{attribute 'linkalways'} 
{attribute 'no_explicit_call' := 'This FB is a CLASS and must be accessed using methods or properties'}
{attribute 'enable_dynamic_creation'}
FUNCTION_BLOCK ReleaseAxisCommand EXTENDS NciCommand
VAR
	_fb : CfgReconfigAxis;
	_axisId : UDINT;
	_timeout : TIME;
END_VAR

METHOD FB_init : BOOL
VAR_INPUT
	bInitRetains : BOOL; // if TRUE, the retain variables are initialized (warm start / cold start)
	bInCopyCode : BOOL;  // if TRUE, the instance afterwards gets moved into the copy code (online change)
	axis : I_Axis;
	timeout : TIME;
END_VAR
IF axis <> 0 THEN
	_axisId := axis.AxisId;
END_IF
_timeout := timeout;
END_METHOD

METHOD PROTECTED  WhileBusy
VAR_INPUT
	CommandState : I_CommandBusyState;
END_VAR
_fb(
	bExecute := TRUE,
	nAxisId := _axisId,
	tTimeOut := _timeout
);

IF _fb.bBusy THEN
	RETURN;
END_IF

IF _fb.bErr THEN
	CommandState.SetError(_fb.nErrId);
	_fb(bExecute := FALSE);
	RETURN;
END_IF

_fb(bExecute := FALSE);
CommandState.SetDone();
END_METHOD

END_FUNCTION_BLOCK

(* stored: Version 1.1.0.1, ProductVersion 3.1.4024.12
   POU ReleaseAxisCommand: Id {1379fa3c-8be3-4107-ae26-0fb3b7f0c80e}, SpecialFunc None
   Method FB_init: Id {df49a14d-365f-4419-b7ca-7a6dafac7a0a}
   Method WhileBusy: Id {82a03946-48f6-4524-b6a0-8325c63f75a4} *)
